# EPICS substitutions: db/Beckhoff_3XXX/ecmcEL3681_ALL.substitutions
file "ecmc_analogInput-chX.template"
{
  pattern {CH_ID, ESLO,         EOFF,      EGU,     PREC}
          {01,    ${ESLO=1E-6}, ${EOFF=0}, ${EGU=}, 6   }
}

file "ecmcEL3681-stat-chX.template"
{
  pattern {CH_ID, KEY }
          {01,    "AI"}
}

file "ecmcEL3681-ModeRange-chX.template"
{
  pattern {CH_ID, KEY }
          {01,    "AI"}
}
